(*
version 1.0	1 sep 2006
programmer 	hugo
tested by		tobias

this function calculates the power equation f_power = a*x^n

*)
FUNCTION F_POWER : REAL
VAR_INPUT
	a : REAL;
	x : REAL;
	n : REAL;
END_VAR

F_POWER := a * EXPT(X, N);

END_FUNCTION

(* stored: Version 1.1.0.1
   POU F_POWER: Id {8f72a1ce-ab59-4091-9c0f-7fefa76001f5}, SpecialFunc None *)
